INTERFACE IAssertionMessageList

METHOD AddMessage : BOOL
VAR_INPUT
    Message : T_MaxString;
END_VAR
END_METHOD

METHOD Clear
VAR_INPUT
END_VAR
END_METHOD

END_INTERFACE

(* stored: Version 1.1.0.1, ProductVersion 3.1.4024.3
   Itf IAssertionMessageList: Id {ff44114b-d9b1-4d5a-96bc-cf1b9c7dac9e}
   Method AddMessage: Id {7cdd12b2-af5d-4c54-bcf4-fc15d1620a8e}
   Method Clear: Id {630af960-6780-4c4e-9e49-9f2fb73a9e7e} *)
